FUNCTION_BLOCK PUBLIC FB_LiveBit
VAR_INPUT
	InTrigger:BOOL;
END_VAR
VAR_OUTPUT
	OutReTrigger:BOOL;
END_VAR
VAR
	m_Tof			:TOF;
	m_PosFlk		:R_TRIG;
	m_NegFlk		:F_TRIG;
	m_Toogle		:BOOL;
	
	m_Counter:INT;
END_VAR

m_PosFlk(CLK:=InTrigger);
m_NegFlk(CLK:=InTrigger);

m_Tof(IN:=m_PosFlk.Q OR m_NegFlk.Q,PT:=T#2S);
IF NOT m_Tof.Q THEN
	m_Toogle:=NOT m_Toogle;
ELSE
	m_Toogle:=FALSE;
END_IF

END_FUNCTION_BLOCK

(* stored: Version 1.1.0.1, ProductVersion 3.1.0.36
   POU FB_LiveBit: Id {37a0ca57-803f-4843-920a-c0fab2481626}, SpecialFunc None *)
